(* CoDeSys 2.3.9.62 project: Tema1 Ejemplo1-Motor v0.pro *)
(* Libraries: Standard.lib 2.6.14 10:37:46 *)

(* POU PLC_PRG, LD *)
PROGRAM PLC_PRG
VAR
	S1: BOOL;
	S2: BOOL;
	Motor: BOOL;
      KM1 :BOOL;
END_VAR
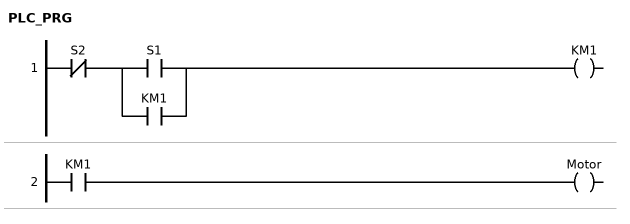
_LD_ (* Ladder Diagram *)
NETWORK 1
	[/S2] - { [S1] | [KM1] } --- (KM1)
NETWORK 2
	[KM1] --- (Motor)
_END_LD_
(* the same logic as Structured Text *)
(* Network 1 *)
KM1 := NOT S2 AND (S1 OR KM1);
(* Network 2 *)
Motor := KM1;
END_PROGRAM

(* Visualisation Botonera
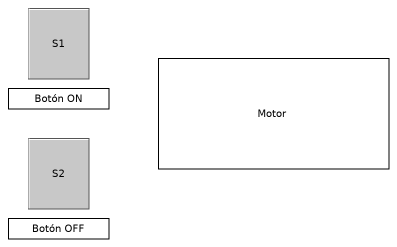
rounded rectangle at (200,80)-(431,191): text "Motor"; shows PLC_PRG.temp1.ET; alarm colour if PLC_PRG.Motor
button at (70,30)-(131,101): text "S1"; taps PLC_PRG.S1
button at (70,160)-(131,231): text "S2"; taps PLC_PRG.S2
rectangle at (50,110)-(151,131): text "Botón ON"
rectangle at (50,240)-(151,261): text "Botón OFF"
*)
